(*

## Short summary

This class provides assert statements for date and time types
It implements `IDateAndTimeAssertions`
For 32 bit date and time types use `DateAndTimeAssertions.simple`
For 64 bit date and time types use `IDateAndTimeAssertions.long`

.. <legal notes>

legal notes
=================
| SPDX-FileCopyrightText: © 2022 ekvip automation GmbH <info@ekvip.de>
| SPDX-License-Identifier: Apache-2.0
| For details check: Apache-2.0_

.. _Apache-2.0: https://www.apache.org/licenses/LICENSE-2.0

.. </legal notes>



*)

{attribute 'reflection'}
FUNCTION_BLOCK INTERNAL DateAndTimeAssertions
EXTENDS CNM_AbstractObject.Object
IMPLEMENTS IDateAndTimeAssertions, IAssertCallBacksetter
VAR
	(* class to handle 32 bit date and time assertions *)
	assertionsFor32BitTypes	:SimpleDateAndTimeAssertions();
	(* class to handle 64 bit date and time assertions *)
	assertionsFor64BitTypes	:LongDateAndTimeAssertions();
END_VAR

(*

## Short summary
This abstract property returns the class name of the concrete object, 
It's for debugging purpose

.. <legal notes>

legal notes
=================
| SPDX-FileCopyrightText: © 2022 ekvip automation GmbH <info@ekvip.de>
| SPDX-License-Identifier: Apache-2.0
| For details check: Apache-2.0_

.. _Apache-2.0: https://www.apache.org/licenses/LICENSE-2.0

.. </legal notes>

*)

PROPERTY className :CNM_AbstractObject.ClassName
GET
className := 'CNM_Assertor.DateAndTimeAssertions';
END_GET
END_PROPERTY

(*

## Short summary
Returns an interface with assert statements for 64 bit times 

.. <legal notes>

legal notes
=================
| SPDX-FileCopyrightText: © 2022 ekvip automation GmbH <info@ekvip.de>
| SPDX-License-Identifier: Apache-2.0
| For details check: Apache-2.0_

.. _Apache-2.0: https://www.apache.org/licenses/LICENSE-2.0

.. </legal notes>

*)

PROPERTY long :ILongDateAndTimeAssertions
GET
long := THIS^.assertionsFor64BitTypes;
END_GET
END_PROPERTY

(*

## Short summary
This methods is the setter for the callback class if an assertion was false

.. <legal notes>

legal notes
=================
| SPDX-FileCopyrightText: © 2022 ekvip automation GmbH <info@ekvip.de>
| SPDX-License-Identifier: Apache-2.0
| For details check: Apache-2.0_

.. _Apache-2.0: https://www.apache.org/licenses/LICENSE-2.0

.. </legal notes>



*)

METHOD setCallBack
VAR_INPUT
	(* the class that must be informed if an assertion is false *)
	callBack	:IAssertCallBack;  
END_VAR
THIS^.assertionsFor32BitTypes.setCallBack(callBack);
THIS^.assertionsFor64BitTypes.setCallBack(callBack);
END_METHOD

(*

## Short summary
Returns the interface `ISimpleDateAndTimeAssertions`
with assert statements for date and time types with 32 bit length

.. <legal notes>

legal notes
=================
| SPDX-FileCopyrightText: © 2022 ekvip automation GmbH <info@ekvip.de>
| SPDX-License-Identifier: Apache-2.0
| For details check: Apache-2.0_

.. _Apache-2.0: https://www.apache.org/licenses/LICENSE-2.0

.. </legal notes>



*)

PROPERTY simple :ISimpleDateAndTimeAssertions
GET
simple := THIS^.assertionsFor32BitTypes;
END_GET
END_PROPERTY

END_FUNCTION_BLOCK

(* stored: Version 1.1.0.1, ProductVersion 3.1.4026.12
   POU DateAndTimeAssertions: Id {53385353-02b0-42a0-b691-66e800470802}, SpecialFunc None
   Property className: Id {11e0bfa9-2ead-4f6b-9b93-22212ea736b0}
   Get Get: Id {343b398a-08c2-4cab-8206-2815786a7725}
   Property long: Id {0835d015-cacc-4bb5-964d-1d1a603d12af}
   Get Get: Id {f7543acb-d3b2-4734-8613-805cb64a45c4}
   Method setCallBack: Id {4e31c649-5f75-4d78-808d-eb927234c3ac}
   Property simple: Id {ce98ce2a-31c2-40d0-8199-146aaf89df45}
   Get Get: Id {6ddc94e8-1ef4-4b5e-b599-a442890025a7} *)
